Staubli VAL3: page_inOut.pjx

--- page_inOut.pjx ---
Parameters version=s7.5 stackSize=5000 millimeterUnit=true
Program file=alreadyExist.pgx
Program file=buildList.pgx
Program file=buildList2.pgx
Program file=insertIO.pgx
Program file=listAdd.pgx
Program file=loadNext.pgx
Program file=main.pgx
Program file=onBackEvent.pgx
Program file=onEnterEvent.pgx
Program file=onExit.pgx
Program file=onF1Event.pgx
Program file=onF2Event.pgx
Program file=onF3Event.pgx
Program file=onF4Event.pgx
Program file=onF5Event.pgx
Program file=onF6Event.pgx
Program file=onF7Event.pgx
Program file=onF8Event.pgx
Program file=onSpaceEvent.pgx
Program file=onStart.pgx
Program file=refresh.pgx
Program file=refreshDynamic.pgx
Program file=refreshStatic.pgx
Program file=showExist.pgx
Data file=page_inOut.dtx
Library alias=page path=Disk://kernel/template/page/page.pjx
Library alias=use path=Disk://kernel/userPage/userPage.pjx
Library alias=language path=Disk://kernel/language/language.pjx
Library alias=saveData path=Disk://saveData/saveData.pjx
Library alias=prog path=Disk://instruction/PROG/PROG.pjx
Library alias=in path=Disk://instruction/inputOutput/IN/IN.pjx
Library alias=out path=Disk://instruction/inputOutput/OUT/OUT.pjx
Library alias=NUM path=Disk://instruction/inputOutput/NUM/NUM.pjx
Library alias=saveInOut path=Disk://saveInputOutput/saveInputOutput.pjx
Type name=InstrItem path=Disk://kernel/template/InstrItem/InstrItem.pjx

--- page_inOut.dtx ---
bool bButton[8]
  [6] = true
  [7] = true
bool bLarge = true
num nIndex
num nInsert
num nKey = -1
public num nPage
num nRefresh
num nSelected = -1
num nTime = 0.5
num nView
num nViewMode = 1
string sEvent
public string sItems
string sList
string sMenu[8]
  [6] = "Delete"
  [7] = "New"
string sMenu8[8]
string sMessage
string sMode = "OUT"
string sId

--- main.pgx ---
public program main()
  local bool l_bSaveInOut
  local bool l_bSaveData
  local bool l_bRefresh
begin
  // INIT
  call onStart()
  // LOOP UNTIL nKey=255
  do
    nKey=getKey()
    call use:listevent(nKey,nIndex,sEvent)
    nView=use:nView
    //
    if sEvent!="" and find(sEvent," {")!=-1 and find(sEvent,"]")!=-1
      sId=left(sEvent,find(sEvent," {"))
      sId=right(sId,len(sId)-find(sId,"]")-2)
    endIf
    //
    switch nKey
      case 259
        // TAB ENLARGE
       // bLarge=!bLarg
        call use:setView(bLarge)
        use:bUseRefresh=true
      break
      case 32
        // ON-OFF
        call onSpaceEvent(sId)
        use:bUseRefresh=true
      break
      case 264
        // left
        nViewMode=(nViewMode+2)%3
        sId=""
        use:bUseRefresh=true
      break
      case 268
        //right
        nViewMode=(nViewMode+1)%3
        sId=""
        use:bUseRefresh=true
      break
      case 271
        if sId!=""
          // Disable-Enable the output
          call onF1Event(sId,l_bSaveInOut)
          l_bSaveInOut=true
        endIf
      break
      case 272
        call onF2Event()
      break
      case 273
        call onF3Event()
      break
      case 274
        call onF4Event()
      break
      case 275
        // SELECT_UNSELECT
        if sId!=""
          call onF5Event(sId,l_bSaveInOut)
          l_bSaveData=true
        endIf
      break
      case 276
        // ON_OFF
        call onF6Event()
      break
      case 277
        // Delete
        if sId!=""
          call onF7Event(sId,l_bSaveInOut)
          l_bSaveInOut=true
          use:bUseRefresh=true
        endIf
      break
      case 278
        // New
        call onF8Event(l_bSaveInOut)
        l_bSaveInOut=true
        use:bUseRefresh=true
      break
      case 270
        // USE ALSO BACKSPACE
        // edit the value ->rename
        if sId!=""
          call onEnterEvent(sId,l_bSaveInOut)
          use:bUseRefresh=true
        endIf
      break
      case 263
        // BACKSPACE
        if sId!=""
          call onBackEvent(sId,l_bSaveInOut)
          use:bUseRefresh=true
        endIf
      break
    endSwitch
    //
    call refresh()
    //release the resource
    delay(0)
  until nKey==255
  // on Exit
  call onExit(l_bSaveInOut,l_bSaveData)
end

--- alreadyExist.pgx ---
program alreadyExist(string& x_sName[], bool& x_bFound[])
  local num l_nResult
  local string l_sMessage
  local string l_sMessage2
  local InstrItem l_iItem
begin
  switch nViewMode
    case 0
      l_iItem.sType="OUT"
    break
    case 1
      l_iItem.sType="IN"
    break
    case 2
      l_iItem.sType="NUM"
    break
  endSwitch
  // set the data
  l_iItem.sData=x_sName
  // search inside all the program - trajectory - tcp
  call prog:findItem(l_iItem,l_nResult,true)
  if l_nResult!=0
    // show the item if it exists
    call showExist(x_sName,sMessage)
    x_bFound=true
  else
    x_bFound=false
  endIf
end

--- buildList.pgx ---
program buildList(num x_nViewMode (dimensions=1))
  local num i
  local string l_sEvent
  local string l_sTemp
  local string l_sId
  local string l_sName
  local bool l_bStatus
  local bool l_bActive
  local string l_sEmpty
  local num l_nSizeOut
  local num l_nSizeIn
  local string l_sMessage
begin
  // INIT the list
  l_sEmpty=""
  l_nSizeOut=-1
  l_nSizeIn=-1
  call out:getSize(l_nSizeOut)
  call in:getSize(l_nSizeIn)
  call use:stringCopy(l_sEmpty,sList)
  // set the view
  switch x_nViewMode
    case 0
      //
      // output
      //
      sMode="OUT"
      for i=0 to l_nSizeOut-1
        // get
        call out:get(l_sId,i)
        call out:isActive(l_bActive,l_sId)
        if l_bActive
          call out:getStatus(l_bStatus,l_sId)
          call use:showBoolStatus(l_bStatus,l_sTemp)
          call out:getItem(l_sName,l_sId)
          call out:isEnable(l_bStatus,l_sId)
          if l_bStatus
            call listAdd(l_sTemp+" "+l_sId+" {"+l_sName+"}")
          else
            call listAdd(l_sTemp+"!"+l_sId+" {"+l_sName+"}")
          endIf
          // SET THE START_STOP_END_HOME
          if l_sName=="start"
            saveData:sOutStart=l_sId
          elseIf l_sName=="stop"
            saveData:sOutStop=l_sId
          elseIf l_sName=="end"
            saveData:sOutEnd=l_sId
          elseIf l_sName=="home"
            saveData:sOutHome=l_sId
          endIf
        endIf
      endFor
    break
    case 1
      //
      // INPUT
      //
      sMode="IN"
      for i=0 to l_nSizeIn-1
        // CS8
        call in:get(l_sId,i)
        call in:isActive(l_bActive,l_sId)
        if l_bActive
          call in:getStatus(l_bStatus,l_sId)
          call use:showBoolStatus(l_bStatus,l_sTemp)
          call in:getItem(l_sName,l_sId)
          call in:isEnable(l_bStatus,l_sId)
          if l_bStatus
            call listAdd(l_sTemp+" "+l_sId+" {"+l_sName+"}")
          else
            call listAdd(l_sTemp+"!"+l_sId+" {"+l_sName+"}")
          endIf
          // SET THE START_STOP_END_HOME
          if l_sName=="start"
            saveData:sInStart=l_sId
          elseIf l_sName=="stop"
            saveData:sInStop=l_sId
          elseIf l_sName=="end"
            saveData:sInEnd=l_sId
          elseIf l_sName=="home"
            saveData:sInHome=l_sId
          endIf
        endIf
      endFor
    break
  endSwitch
  // rebuild the Function LIST
  call use:listempty()
  call use:listadd(sList)
end

--- buildList2.pgx ---
program buildList2(num x_nViewMode)
  local num l_nSize
  local num i
  local string l_sName
  local bool l_bActive
  local num l_nValue
  local string l_sEmpty
  local string l_sField
  local string l_sItem
begin
  // INIT the list
  l_sEmpty=""
  call use:stringCopy(l_sEmpty,sList)
  // get the size
  call NUM:getSize(l_nSize)
  // Build the list
  for i=0 to l_nSize-1
    call NUM:get(l_sItem,i)
    call saveInOut:getItem_num(l_sName,l_sItem)
    call NUM:isActive(l_bActive,l_sItem)
    if l_bActive
      call saveInOut:getValue_num(l_nValue,l_sItem)
      // COUNTING
      call listAdd("["+toString("3",l_nValue)+"] "+l_sItem+" {"+l_sName+"}")
    endIf
  endFor
  // rebuild the list
  call use:listempty()
  call use:listadd(sList)
end

--- insertIO.pgx ---
program insertIO(num& x_nIndex[])
  local string l_sMessage
  local bool bActive
  local num l_nSizeIn
  local num l_nSizeOut
  local string l_sItem
  local num i
  local string l_sKey
  local string l_sStatus
  local bool l_bStatus
  local num l_nSelect
  local bool l_bInsert
begin
  // create the list
  call use:setSizeList(14,0,19,11)
  call use:clear(0,13)
  call language:message(l_sMessage,65)
  call use:typeCenter(13,l_sMessage,40,true)
  // get the value
  call in:getSize(l_nSizeIn)
  call out:getSize(l_nSizeOut)
  switch nViewMode
    case 0
      //
      // OUTPUT
      //
      call use:listcreate("")
      for i=0 to l_nSizeOut-1
        call out:get(l_sKey,i)
        call out:getItem(l_sItem,l_sKey)
        call out:isActive(l_bStatus,l_sKey)
        if !l_bStatus
          l_sMessage=l_sKey+"{"+l_sItem+"}"
          call use:listadd(l_sMessage)
          l_bInsert=true
        endIf
      endFor
      // list update
      call use:listupdate(min(nInsert,l_nSizeOut))
    break
    case 1
      //
      // INPUT
      //
      call use:listcreate("")
      for i=0 to l_nSizeIn-1
        call in:get(l_sKey,i)
        call in:getItem(l_sItem,l_sKey)
        call in:isActive(l_bStatus,l_sKey)
        if !l_bStatus
          l_sMessage=l_sKey+"{"+l_sItem+"}"
          call use:listadd(l_sMessage)
          l_bInsert=true
        endIf
      endFor
      // list update
      call use:listupdate(min(nInsert,l_nSizeIn))
    break
  endSwitch
  if l_bInsert
    // Select ???
    do
      nKey=get()
      call use:listevent(nKey,nInsert,l_sItem)
      // release the resource
      if nKey==270 and l_sItem!=""
        l_sItem=left(l_sItem,find(l_sItem,"{"))
        switch nViewMode
          case 0
            // OUTPUT
            call out:setActive(true,l_sItem)
          break
          case 1
            // INPUT
            call in:setActive(true,l_sItem)
          break
        endSwitch
        // exit
        return
      endIf
    until nKey==255
  endIf
  call use:nullKey(nKey)
end

--- listAdd.pgx ---
program listAdd(string x_sEvent (dimensions=1))
begin
  // add in the queue
  if sList!=""
    insert(sList[size(sList)])
  endIf
  sList[size(sList)-1]=x_sEvent
end

--- loadNext.pgx ---
program loadNext(string x_sPage, string& x_sItems[])
// load the next page
  local num i
  local string l_sMessage
begin
  // look if the page libload is correct
  i=page:libLoad(x_sPage)
  delay(0)
  if i!=0
    logMsg("[KERNEL] INTERFACE:PAGE LIBLOAD "+x_sPage+" result "+toString("",i))
    call language:message(l_sMessage,-7)
    popUpMsg(l_sMessage+x_sPage+" ; "+toString("",i))
  else
    // copy all the field from x_sItems to the next page
    call use:stringCopy(x_sItems,page:sItems)
    call page:main()
  endIf
end

--- onBackEvent.pgx ---
program onBackEvent(string x_sId, bool& x_bSave[])
  local bool l_bFound
  local num l_nX
  local num l_nY
  local string l_sString
  local string l_sMessage
  local bool l_bOk
  local num l_nValue
begin
  //
  // NB sEvent is the selected
  // element in the LIST
  //
  switch nViewMode
    case 0,1
      // OUT IN NUM
      call onEnterEvent(x_sId,x_bSave)
    break
    case 2
      // COUNT
      l_nX=40-use:nBottomX+find(sEvent,"{")
      call saveInOut:getItem_num(l_sString,x_sId)
      l_nY=nView+1
      // clean the line
      call use:listcursor(use:nView,false)
      // read the name
      call use:read(l_nX,l_nY,l_sString,14,false)
      // check if already exist
      if !use:bUseEscape and l_sString!=""
        // set the value
        call NUM:set(l_sString,x_sId)
      endIf
      // save it
      x_bSave=true
    break
  endSwitch
end

--- onEnterEvent.pgx ---
program onEnterEvent(string x_sId, bool& x_bSave[])
  local bool l_bFound
  local num l_nX
  local num l_nY
  local string l_sString
  local string l_sMessage
  local bool l_bOk
  local num l_nValue
  local string l_sName
begin
  //
  // NB sEvent is the selected
  // element in the LIST
  //
  l_nX=40-use:nBottomX+find(sEvent,"{")
  // select
  switch nViewMode
    case 0
      // OUT
      call out:getItem(l_sString,x_sId)
    break
    case 1
      // IN
      call in:getItem(l_sString,x_sId)
    break
    case 2
      // COUNT
      call saveInOut:getItem_num(l_sString,x_sId)
    break
  endSwitch
  // set the list
  l_nY=nView+1
  if nViewMode!=2
    // clean the line
    call use:listcursor(use:nView,false)
  endIf
  // read the name
  l_sName=l_sString
  call use:read(l_nX,l_nY,l_sString,14,false)
  // check if already exist
  if !use:bUseEscape and l_sString!=l_sName and l_sString!=""
    switch nViewMode
      case 0
        // OUT
        call out:setItem(l_sString,x_sId)
      break
      case 1
        // IN
        call in:setItem(l_sString,x_sId)
      break
      case 2
        // COUNT
        call NUM:set(l_sString,x_sId)
      break
    endSwitch
    // save it
    x_bSave=true
  endIf
end

--- onExit.pgx ---
program onExit(bool x_bSaveInOut (dimensions=1), bool x_bsaveData (dimensions=1))
  local num l_nResult
  local string l_sMessage
begin
  // SAVE IT
  if x_bSaveInOut
    call out:save(l_nResult)
    if l_nResult!=0
      call language:message(l_sMessage,-6)
      popUpMsg(l_sMessage+toString("",l_nResult))
      logMsg("[KERNEL] INTERFACE:Error saving Out code: "+toString("",l_nResult))
    else
    endIf
    call in:save(l_nResult)
    if l_nResult!=0
      call language:message(l_sMessage,-6)
      popUpMsg(l_sMessage+toString("",l_nResult))
      logMsg("[KERNEL] INTERFACE:Error saving In code: "+toString("",l_nResult))
    endIf
    // save all the data
    if x_bsaveData
      l_nResult=saveData:libSave()
      if l_nResult!=0
        call language:message(l_sMessage,-6)
        popUpMsg(l_sMessage+toString("",l_nResult))
        logMsg("[KERNEL] INTERFACE:Error saving saveData code: "+toString("",l_nResult))
      endIf
    endIf
  endIf
  // clear the list
  call use:listempty()
end

--- onF1Event.pgx ---
program onF1Event(string x_sItem (dimensions=1), bool& x_bSave[] (dimensions=1))
  local bool l_bChange
  local bool l_bStatus
begin
  // look if the bButton is enable
  if bButton[0]
    if sMode=="OUT"
      // OUTPUT
      call out:isEnable(l_bStatus,x_sItem)
      call out:setEnable(!l_bStatus,x_sItem)
      logMsg("[KERNEL] INTERFACE:Change the active status of: "+x_sItem)
    elseIf sMode=="IN"
      // INPUT
      call in:isEnable(l_bStatus,x_sItem)
      call in:setEnable(!l_bStatus,x_sItem)
      logMsg("[KERNEL] INTERFACE:Change the active status of: "+x_sItem)
    endIf
    // save it
    x_bSave=true
  endIf
end

--- onF5Event.pgx ---
program onF5Event(string x_sId, bool& x_bSave[])
  local string l_sMessage
  local num lKey
  local num i
  local string l_sItem
  local num l_nSize
  local bool l_bFound
  local string l_sEmpty
  local string l_sName
begin
  // look if the bButton is enable
  if bButton[4]
    //
    if sMode=="OUT"
      //
      // OUTPUT FUNCTION
      //
      call out:getItem(l_sName,x_sId)
      if l_sName!="start" and l_sName!="stop" and l_sName!="end" and l_sName!="home"
        call use:setSizeList(10,1,15,9)
        call use:listcreate("")
        l_sItem="start"
        call use:listadd(l_sItem)
        l_sItem="stop"
        call use:listadd(l_sItem)
        l_sItem="end"
        call use:listadd(l_sItem)
        l_sItem="home"
        call use:listadd(l_sItem)
        call use:listupdate(0)
        call use:clear(0,13)
        do
          lKey=get()
          call use:listevent(lKey,i,l_sItem)
        until lKey==255 or lKey==270
        if lKey==270
          // LOOK IF EXIST
          call out:find(l_sItem,l_bFound)
          if !l_bFound
            call out:setItem(l_sItem,x_sId)
            x_bSave=true
          endIf
          if l_bFound
            // ALREADY EXIST
            call language:message(l_sMessage,-2)
            popUpMsg(l_sMessage)
          endIf
        else
          // release the Key
          call use:nullKey(lKey)
        endIf
      else
        // restore the old_Name
        call out:setItem(x_sId,x_sId)
        x_bSave=true
      endIf
    elseIf sMode=="IN"
      //
      // INPUT FUNCTION
      //
      call in:getItem(l_sName,x_sId)
      if find(sEvent,"#")==-1 and l_sName!="start" and l_sName!="stop" and l_sName!="end" and l_sName!="home"
        call use:setSizeList(10,1,15,9)
        call use:listcreate("")
        call prog:getSize(l_nSize)
        l_sItem=" ---PROG ---------- "
        call use:listadd(l_sItem)
        for i=0 to l_nSize-1
          call prog:get(l_sItem,i)
          if l_sItem!="" and find(l_sItem,"#")!=-1
            call use:listadd(l_sItem)
          endIf
        endFor
        l_sItem=" ------------------ "
        call use:listadd(l_sItem)
        l_sItem="start"
        call use:listadd(l_sItem)
        l_sItem="stop"
        call use:listadd(l_sItem)
        l_sItem="end"
        call use:listadd(l_sItem)
        l_sItem="home"
        call use:listadd(l_sItem)
        //
        call use:listupdate(0)
        call language:message(l_sMessage,60)
        call use:type(1,13,l_sMessage)
        do
          lKey=get()
          call use:listevent(lKey,i,l_sItem)
        until lKey==255 or lKey==270
        if lKey==270 and find(l_sItem,"------")==-1
          if l_sItem!="start" and l_sItem!="stop" and l_sItem!="end" and l_sItem!="home"
            logMsg("[KERNEL] INTERFACE:Associate the program: "+l_sItem+" to: "+sEvent)
          endIf
          // LOOK IF EXIST
          call in:find(l_sItem,l_bFound)
          if !l_bFound
            call in:setItem(l_sItem,x_sId)
            x_bSave=true
          endIf
          if l_bFound
            // ALREADY EXIST
            call language:message(l_sMessage,-2)
            popUpMsg(l_sMessage)
          endIf
        else
          // release the Key
          call use:nullKey(lKey)
        endIf
      else
        // restore the old_Name
        call in:setItem(x_sId,x_sId)
        x_bSave=true
      endIf
    endIf
  endIf
  // check if to reload all
  if x_bSave
    saveData:bChangeIO=true
  endIf
end

--- onF6Event.pgx ---
program onF6Event()
  local bool l_bStatus
begin
  // look if the bButton is enable
  if bButton[5]
  endIf
end

--- onF7Event.pgx ---
program onF7Event(string x_sId (dimensions=1), bool x_bSave (dimensions=1))
  local string l_sName
  local num i
  local num l_nResult
  local bool l_bFound
  local string l_sButton[2]
  local string l_sMessage
  local bool l_bYes
begin
  // look if the bButton is enable
  if bButton[6]
    //
    // DELETE
    //
    if sMode=="IN" and find(sEvent,"usr")==-1 and find(sEvent,"fast")==-1
      // compose the search "IN,l_sName"
      call alreadyExist(x_sId,l_bFound)
      // if not found
      if !l_bFound
        call language:message(l_sMessage,22)
        // get the yes_no button Key
        call language:getYesNo(l_sButton)
        // ask the question
        call use:yes_no(l_sMessage+sEvent,l_sButton,l_bYes)
        if l_bYes
          call in:setActive(false,x_sId)
          logMsg("[KERNEL] INTERFACE:Disable the Input: "+l_sName)
          x_bSave=true
        endIf
      endIf
    elseIf sMode=="OUT" and find(sEvent,"valve")==-1 and find(sEvent,"fast")==-1
      call alreadyExist(x_sId,l_bFound)
      // if not found
      if !l_bFound
        call language:message(l_sMessage,22)
        // get the yes_no button Key
        call language:getYesNo(l_sButton)
        // ask the question
        call use:yes_no(l_sMessage+sEvent,l_sButton,l_bYes)
        if l_bYes
          call out:setActive(false,x_sId)
          logMsg("[KERNEL] INTERFACE:Disable the Output: "+l_sName)
          x_bSave=true
        endIf
      endIf
    endIf
    // scan the system
    if l_nResult!=0
      // show that the item already exist
      call showExist(l_sName,sMessage)
    endIf
  endIf
end

--- onF8Event.pgx ---
program onF8Event(bool& x_bSave[] (dimensions=1))
begin
  // look if the bButton is enable
  if bButton[7]
    //
    call insertIO(nSelected)
    x_bSave=true
  endIf
end

--- onSpaceEvent.pgx ---
program onSpaceEvent(string x_sId)
  local bool l_bStatus
  local num l_nX
  local num l_nValue
  local string l_sString
  local num l_nY
  local bool l_bOk
begin
  //
  // NB sEvent is the selected
  // element in the LIST
  //
  //
  if nViewMode==0
    call out:getStatus(l_bStatus,x_sId)
    call out:setStatus(!l_bStatus,x_sId)
    logMsg("[KERNEL] INTERFACE:Change the status ON/OFF of: "+sEvent)
  elseIf nViewMode==2
    if find(x_sId,"In")!=-1
      // INPUT not allowed
      return
    else
      l_nX=40-use:nBottomX+find(sEvent,"[")
      call saveInOut:getValue_num(l_nValue,x_sId)
      l_sString=toString("3",l_nValue)
    endIf
    // set IT
    l_nY=nView+1
    call use:read(l_nX,l_nY,l_sString,14,false)
    // COUNT
    toNum(l_sString,l_nValue,l_bOk)
    if l_bOk
      // set the value
      call NUM:setValue(l_nValue,x_sId)
    endIf
  endIf
end

--- onStart.pgx ---
program onStart()
  local num i
  local bool bTest
begin
  // logMsg
  logMsg("[KERNEL] INTERFACE:PAGE Input Output")
  //
  sMode="OUT"
  sId=""
  nViewMode=0
  // refresh all
  call refreshStatic()
  call buildList(0)
  // record the old value....
  call use:selectNewField(nSelected,nIndex,nView)

end

--- refresh.pgx ---
program refresh()
// page refresh
begin
  //
  // refresh the static message
  if (nKey>270 and nKey<=278) or (nKey==259 or nKey==264 or nKey==268) or use:bUseRefresh
    call refreshStatic()
    call refreshDynamic()
  else
    // refresh the Dynamic message
    if abs(clock()-nRefresh)>nTime
      call refreshDynamic()
    endIf
  endIf
end

--- refreshDynamic.pgx ---
program refreshDynamic()
  local bool l_bStatus
  local bool l_bReserved
  local string l_sMessage
  local string l_sEmpty
begin
  // DO NOT CHANGE
  nRefresh=clock()
  use:bUseRefresh=false
  // update the list
  if nViewMode==2
    // show the count list
    call buildList2(nViewMode)
  else
    // build the list
    call buildList(nViewMode)
  endIf
  //
  // ADD HERE
  //
  // this function ables to set the ON/OFF when you focus an OUT
  // or SELECT/UNSELECT a program if is an INPUT
  //
  //
  // SET THE PAGE NUMBER
  use:nPage=110
  // USE <> PROFILE for <> PAGE
  use:nPage=use:nPage+abs(limit(saveData:mode,0,2)-2)
  // get the data
  if find(sEvent,"start")!=-1 or find(sEvent,"stop")!=-1 or find(sEvent,"end")!=-1 or find(sEvent,"home")!=-1 or find(sEvent,"*")!=-1
    l_bReserved=true
  endIf
  // check th sID
  if sId!=""
    switch nViewMode
      case 0
        call out:isEnable(l_bStatus,sId)
      break
      case 1
        call in:isEnable(l_bStatus,sId)
      break
      case 2
        call use:stringCopy(l_sEmpty,sMenu)
      break
    endSwitch
  endIf
  if nViewMode==0 or nViewMode==1
    // show the menu
    if saveData:language!="japanese"
      // SET THE VIEW OF THE PAGE
      call language:page(l_sMessage,use:nPage)
      // define the menu
      call use:stringToArray(l_sMessage,sMenu)
      // show the F1 - F5 button
      if l_bStatus or sId==""
        call language:message(l_sMessage,38)
      else
        call language:message(l_sMessage,37)
      endIf
      sMenu[0]=l_sMessage
      if !l_bReserved
        call language:message(l_sMessage,35)
      else
        call language:message(l_sMessage,36)
      endIf
      // activate the option button F5
      if size(sMenu)>5
        sMenu[4]=l_sMessage
      endIf
      if !bLarge
        call use:setMenu(sMenu,true,3)
      else
        call use:setMenu(sMenu,true,-1)
      endIf
    else
      // japanese use the array for the menu
      call language:page(sMenu8,use:nPage)
      call use:stringCopy(sMenu8,sMenu)
      // show the F1 - F5 button
      if !l_bStatus
        sMenu8[0]="Enable"
      else
        sMenu8[0]="Disable"
      endIf
      if !l_bReserved
        sMenu8[4]="Select"
      else
        sMenu8[4]="Unselect"
      endIf
      if !bLarge
        call use:setMenu(sMenu8,false,3)
      else
        call use:setMenu(sMenu8,false,-1)
      endIf
    endIf
  endIf
  // refresh it
  call use:getMenu(sMenu,bButton)
  //bButton[0]=true
  // refresh the list
  call use:selectNewField(nSelected,nIndex,nView)
  nSelected=-1
end

--- refreshStatic.pgx ---
program refreshStatic()
  local num l_nLocal
  local string l_sMessage
begin
  //
  // CREATE THE LIST
  // define your list size for default
  //
  cls()
  call use:setSizeList(19,0,19,11)
  call use:setView(bLarge)
  //
  switch nViewMode
    case 0
      call use:listcreate(" OUT ")
    break
    case 1
      call use:listcreate(" IN ")
    break
    case 2
      call use:listcreate("COUNT")
    break
  endSwitch
  //

end

--- showExist.pgx ---
program showExist(string x_sName (dimensions=1), string x_sMessage (dimensions=1))
  local string l_sMessage
  local string l_sMessage2
begin
  // not possibile to delete rename
  call language:message(l_sMessage,23)
  call language:message(l_sMessage2,29)
  l_sMessage=l_sMessage+x_sName
  popUpMsg(l_sMessage+l_sMessage2+x_sMessage)
end
